PROGRAM MAIN
VAR
	bottone:BOOL:=FALSE;
	c:INT:=0;
END_VAR

IF(bottone= true) THEN
	c:=c+1;
END_IF

END_PROGRAM

(* stored: Version 1.1.0.1
   POU MAIN: Id {9a1d7829-2361-4322-8eee-e0f95c169571}, SpecialFunc None *)
